# EPICS substitutions: MDrive/motor.substitutions
# ImsMDrivePlus asyn model 3 substitutions file

# SREV (not shown) is the number of steps per revolution is 200 by
#    default
#
# There are three pivot points to which the six motors are attached.
# Three provide vertical motion: M0Y, M1Y, and M2Y.  One provides
# horizontal motion in the Z direction (along beamline): M2Z.  Two
# provide horizontal motion in the X direction (perpendicular to
# beamline): M0X, M2X.
#

#

# For SREV:
#    2048 = internal encoder (EQ)
#     250 = external encoder, NUMERIK-JENA
#     200 = external encoder, Renishaw
#   51200 = no encoder

# CXI DG4 Support Motion Stand (DG4) Substitution file

file "$(MOTOR)/db/basic_asyn_motor.db"
{
pattern
{P,    N, M, DTYP,         PORT, DESC,       ADDR, EGU, DIR,  VELO, VBAS,  ACCL, BDST, BVEL,  BACC, DHLM, DLLM, MRES,     PREC, INIT}
{BL172:MDrive:, 1, m1, "asynMotor",  IMS1, "hx", 0,    mm,  Pos,  0.5,  0.017, 1.0,  0,    0.017, 2.0,  10,  -10, 0.00004, 5,    ""}
{BL172:MDrive:, 1, m2, "asynMotor",  IMS2, "hy", 0,    mm,  Pos,  0.5,  0.017, 1.0,  0,    0.017, 2.0,  18,  3.001, 0.0000083, 5,    ""}
{BL172:MDrive:, 1, m3, "asynMotor",  IMS3, "hz", 0,    mm,  Pos,  0.5,  0.017, 1.0,  0,    0.017, 2.0,  10,  -10, 0.00004, 5,    ""}
{BL172:MDrive:, 1, m4, "asynMotor",  IMS4, "halpha", 0,    deg,  Pos,  0.5,  0.017, 1.0,  0,    0.017, 2.0,  12,  -12, 0.0000125, 5,    ""}
}

file "$(MOTOR)/modules/motorIms/iocs/imsIOC/db/IMS_extra.db"
{
pattern
{DEV, AREA, LOC, PORT, ADDR, TIMEOUT}
{BL172:MDrive:, IOC,    1, IMS1, 0,    1}
{BL172:MDrive:, IOC,    1, IMS2, 0,    1}
{BL172:MDrive:, IOC,    1, IMS3, 0,    1}
{BL172:MDrive:, IOC,    1, IMS4, 0,    1}
}
#       field(DESC,"Y DG4 DS North Motor")  # same
#        field(DTYP,"ImsMDrivePlus")        # same
#        field(OUT, "#C0 S0 @")             # same
#        field(DIR, "Pos")                  # same
#        field(SREV,"2048")                 # SREV [steps/rev], MRES = UREV/SREV
#        field(UREV,"0.017")                # UREV [egu/rev], MRES = UREV/SREV
#        field(UEIP,"No")
#        field(S,   "10")                   # no equivalent
#        field(SMAX,"20")                   # SMAX[rev/s], VELO = SMAX * UREV
#        field(SBAS,"1")                    # VBAS = SBAS * UREV
#        field(ACCL,"2.0")                  # same
#        field(BDST,"0")                    # same
#        field(RDBD,"0.0005")
#        field(RTRY,"1")
#        field(SBAK,"1")                    # BVEL = SBAK * UREV
#        field(BACC,"2.0")                  # same
#        field(DLY, "0")
#        field(PREC,"4")                    # same
#        field(EGU, "mm")                   # same
#        field(DHLM,"200.0")                # same
#        field(DLLM,"-200.0")               # same
#        field(INIT,"")                     # same
#        field(TWV, "1")                    # same
